TYPE EL1xx2_Data :
STRUCT
	{attribute addProperty Name "Channel 1"}
	_1 :DiChannel;
	{attribute addProperty Name "Channel 2"}
	_2 :DiChannel;
END_STRUCT
END_TYPE

(* stored: Version 1.1.0.1, ProductVersion 3.1.4024.9
   DUT EL1xx2_Data: Id {5b835cf4-45e0-0fd9-0660-846b457ae256} *)
